// TIA Portal V17 export
// export: Created 2025-06-26T06:49:16.9635174Z, ExportSetting WithDefaults, DisplayName Totally Integrated Automation Portal, DisplayVersion V17 Update 8, DisplayName TIA Portal Openness, DisplayVersion V17 Update 8, DisplayName TIA Portal Version Control Interface, DisplayVersion V17, DisplayName STEP 7 Professional, DisplayVersion V17 Update 8, DisplayName STEP 7 Safety, DisplayVersion V17 Update 6, DisplayName WinCC Advanced, DisplayVersion V17 Update 8
FUNCTION_BLOCK "fbHysteresis2"   // FB64, LAD
TITLE = fbHysteresis2
{ S7_Optimized_Access := 'TRUE' }
AUTHOR : Heaten
VERSION : 0.1
// Hysteresis function with bool inputs
// stored: AutoNumber true, IsIECCheckEnabled false, IsRetainMemResEnabled false, MemoryReserve 0, SetENOAutomatically false, UDAEnableTagReadback false
   VAR_INPUT
      bEnable : Bool;
      bHigh : Bool;
      bLow : Bool;
      bAbove : Bool;
      bReset : Bool;
   END_VAR
   VAR_OUTPUT
      bOut : Bool;
   END_VAR
   VAR
      State : Bool;
   END_VAR
   VAR_TEMP
      bStartSignal : Bool;
      bStopSignal : Bool;
   END_VAR
BEGIN

REGION Network 1 (SCL): Polarity of the control
   // Above = 1: when process state is "high" eg cooling, emptying, depressurizing
   // Above = 0: when precess state is "low" eg heating, filling, pressurizing
   IF #bAbove = TRUE THEN
       // emptying, cooling, depressurizing etc
       #bStartSignal := #bHigh;
       #bStopSignal := NOT(#bLow);
   ELSE
       // filling, heating, pressurizing etc
       #bStartSignal := NOT(#bLow);
       #bStopSignal := #bHigh;
   END_IF;
END_REGION

REGION Network 2: Switch ouput
   // Initial state = OFF
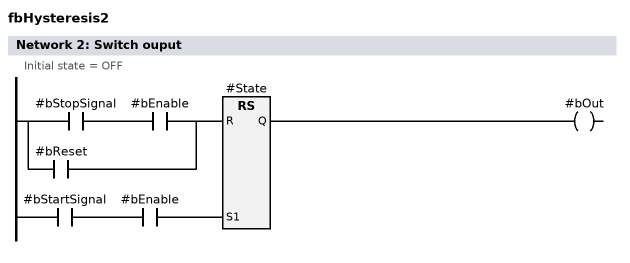
   RUNG wire#powerrail
      Contact( #bStopSignal )
      Contact( #bEnable )
      wire#w1
      S_RS(operand := #State, s1 := wire#w2)
      Coil( #bOut )
   END_RUNG
   RUNG wire#powerrail
      Contact( #bReset )
   END_RUNG wire#w1
   RUNG wire#powerrail
      Contact( #bStartSignal )
      Contact( #bEnable )
   END_RUNG wire#w2
   // the same network as SCL:
   IF (#bStopSignal AND #bEnable) OR #bReset THEN
       #State := FALSE;   // RS flip-flop
   END_IF;
   IF #bStartSignal AND #bEnable THEN #State := TRUE; END_IF;
   #bOut := #State;
END_REGION
END_FUNCTION_BLOCK
